// TIA Portal V18 export
// export: Created 2026-06-22T11:43:40.3118471Z, ExportSetting WithDefaults, DisplayName Totally Integrated Automation Portal, DisplayVersion V18, DisplayName TIA Portal Openness, DisplayVersion V18, DisplayName TIA Portal Version Control Interface, DisplayVersion V18, DisplayName STEP 7 Professional, DisplayVersion V18, DisplayName STEP 7 Safety, DisplayVersion V18, DisplayName WinCC Professional, DisplayVersion V18
Screen "Login/out"  1440x900, Number=1
  ScreenLayer 
    GraphicView "Graphic view_1" at 0,0 size 1440x900  Picture=Thiết kế chưa có tên (1)
    Button "Btn_Login" at 151,156 size 650x85  Mode=Text, StyleItem=Button, TextOff="ĐĂNG NHẬP (LOGIN)", TextOn="Text"
      VisibilityAnimation "VisibilityAnimation"
        tag Logged_In
      on Click: ShowLogonDialog()
    Button "Btn_Logout" at 150,269 size 650x85  Mode=Text, StyleItem=Button, TextOff="ĐĂNG XUẤT (LOGOFF)", TextOn="Text"
      VisibilityAnimation "VisibilityAnimation"  RangeEnd=99, RangeStart=1
        tag Logged_In
      on Click: Logoff()
    Button "Btn_Exit" at 151,411 size 650x85  Mode=Text, StyleItem=Button, TextOff="THOÁT HỆ THỐNG (EXIT)", TextOn="Text"
      on Click: StopRuntime(Mode := 0)
    Button "Btn_Enter_System" at 263,563 size 398x61  Mode=Text, StyleItem=Button, TextOff="VÀO HỆ THỐNG (SCADA)", TextOn="Text"
      VisibilityAnimation "VisibilityAnimation"  RangeEnd=99, RangeStart=1
        tag Logged_In
      on Click: ActivateScreen(Screen name := Man Tong Quan, Object number := 0)
